# EPICS substitutions: src/main/epics/tspd-adqApp/Db/ADQDevice.substitutions
file db/ADQDevice.template {
    pattern { PREFIX, INFO, CHGR, CH }
            { ADQ06215, INFO, AI, CH0 }
            { ADQ06215, INFO, AI, CH1 }
            { ADQ06215, INFO, AI, CH2 }
            { ADQ06215, INFO, AI, CH3 }
}
